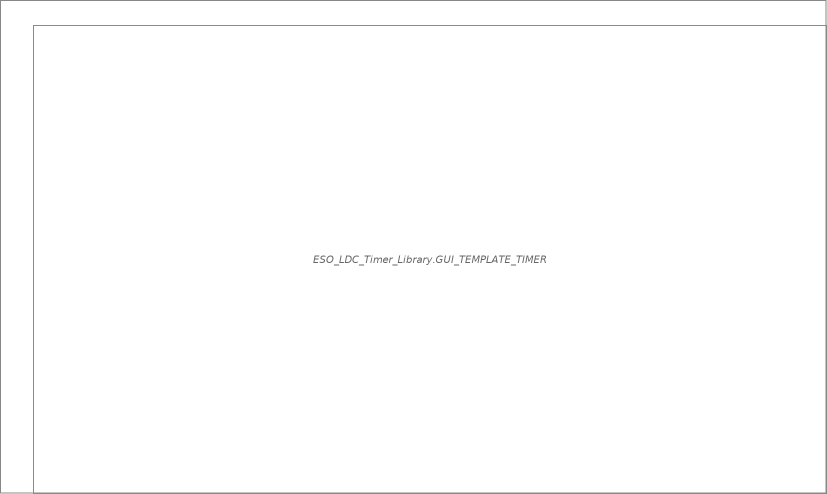
VISUALIZATION GUI_TIMER  // 827x494
    Frame (33,25 794x469)
        shows ESO_LDC_Timer_Library.GUI_TEMPLATE_TIMER(m_Instance := MAIN.fbTimerObj)
END_VISUALIZATION

(* stored: Version 1.1.0.1, ProductVersion 3.1.4024.11
   Visu GUI_TIMER: Id {35fb3887-b26b-4a4f-8ec9-ccb8f09ebf28} *)
